{attribute addProperty BoxType "EJ7031-0000-0026"}
{attribute addProperty Id "ENC_Status_compactAT %I*ENC_Status_compact_FA080ECA4860STM_StatusAT %I*STM_Status_64D937431620ENC_Control_compactAT %Q*ENC_Control_compact_5C86AA9D3240STM_ControlAT %Q*STM_Control_6F24B2C41620STM_VelocityAT %Q*STM_Velocity_1D89B5C21620WcStateAT %I*WcState_98A4DF7520.250InfoDataAT %I*InfoData_1C46E3E796120"}
{attribute addProperty CRC "1132355663"}
{attribute addProperty SizeInBites "226"}
{attribute addProperty SizeInBytes "28.25"}
TYPE EJ7031_26D83138 :
STRUCT
	{attribute addProperty Name "ENC_Status_compact"}
	ENC_Status_compact : ENC_Status_compact_FA080ECA;
	{attribute addProperty Name "STM_Status"}
	STM_Status : STM_Status_64D93743;
	{attribute addProperty Name "ENC_Control_compact"}
	ENC_Control_compact : ENC_Control_compact_5C86AA9D;
	{attribute addProperty Name "STM_Control"}
	STM_Control : STM_Control_6F24B2C4;
	{attribute addProperty Name "STM_Velocity"}
	STM_Velocity : STM_Velocity_1D89B5C2;
	{attribute addProperty Name "WcState"}
	WcState : WcState_98A4DF75;
	{attribute addProperty Name "InfoData"}
	InfoData : InfoData_1C46E3E7;
END_STRUCT
END_TYPE

(* stored: Version 1.2.0.0, ProductVersion 3.1.4024.9
   DUT EJ7031_26D83138: Id {902ef937-0870-463a-bd88-b32c61780426} *)
